(* IEC 61131-3 sources: Std_PalletMover/Class/InterfaceAuxHmiMqtt, 1 file *)

(* ---- InterfaceAuxHmiMqtt.st ---- *)
(*!
<Class
	Name               = "InterfaceAuxHmiMqtt"
	Revision           = "0.0"
	RealtimeTask       = "false"
	CyclicTask         = "false"
	BackgroundTask     = "false"
	Sigmatek           = "false"
	OSInterface        = "false"
	HighPriority       = "false"
	Automatic          = "false"
	UpdateMode         = "Prescan"
	SharedCommandTable = "true"
	Objectsize         = "(810,120)">
	<Channels>
	</Channels>
	<Network Name="InterfaceAuxHmiMqtt">
		<!-- List of Components in this network -->
		<Components>
			<Object
				Name       = "_base"
				Class      = "I_Hmi"
				Position   = "(218,120)"
				Visualized = "false">
				<Channels>
					<Server Name="ClassSvr"/>
				</Channels>
			</Object>
		</Components>
		<Comments>
		</Comments>
		<!-- List of Connections in this network -->
		<Connections>
			<Connection Source="this.ClassSvr" Destination="_base.ClassSvr" Vertices="(1426,210),(1254,210),"/>
		</Connections>
		<!-- Headerfiles -->
		<Options>
		</Options>
	</Network>
</Class>
*)
#pragma using I_Hmi

InterfaceAuxHmiMqtt : CLASS
: I_Hmi
  //Servers:
  //Clients:
  //Variables:
  //Functions:
  //Tables:
	FUNCTION @STD
		VAR_OUTPUT
			ret_code	: CONFSTATES;
		END_VAR;
	FUNCTION GLOBAL TAB @CT_;
END_CLASS;
